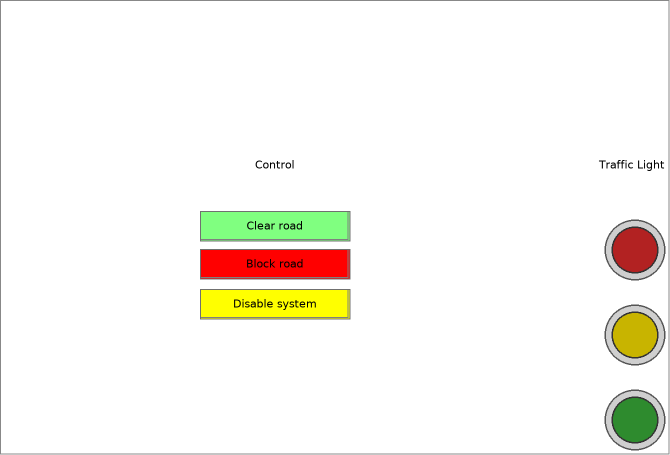
VISUALIZATION VISU_TrafficLight  // 670x455
    Button (200,211 150x30), "Clear road"
        tap MAIN.clear
    Button (200,249 150x30), "Block road"
        tap MAIN.block
    Button (200,289 150x30), "Disable system"
        toggle MAIN.disable
    Lamp1 (600,215 70x70), variable: MAIN.red, style: Lamp-Lamp1-Red
    Lamp1 (600,300 70x70), variable: MAIN.yellow, style: Lamp-Lamp1-Yellow
    Lamp1 (600,385 70x70), variable: MAIN.green, style: Lamp-Lamp1-Green
    Label (600,150 64x30), "Traffic Light"
    Label (200,150 150x30), "Control"
END_VISUALIZATION

(* stored: Version 1.1.0.1, ProductVersion 3.1.4024.9
   Visu VISU_TrafficLight: Id {f0fd67c2-c2c6-4e66-b167-64b049b64f41} *)
